{attribute 'linkalways'} 
{attribute 'no_explicit_call' := 'This FB is a CLASS and must be accessed using methods or properties'}
{attribute 'enable_dynamic_creation'}
FUNCTION_BLOCK Node_F_VN_ReadBarcodeExp2 EXTENDS VisionNode
VAR
    ipSrcImage : _ITcVnImage;
    ipDecodedData : _ITcVnContainer;
	ipContours : _ITcVnContainer;
    eBarcodeType : _ETcVnBarcodeType(ETcVnBarcodeType.TCVN_BT_ANY);
	nCodeNumber : _DINT(1);
	eSearchDirection : _ETcVnBarcodeSearchDirection(ETcVnBarcodeSearchDirection.TCVN_BSD_ANY);
	ipAngles : _ITcVnContainer; 
    hrPrev : _HRESULT(S_OK);
	hresult : _HRESULT(S_OK);
END_VAR

METHOD PUBLIC  Clone : I_Node
VAR
	pNode : POINTER TO Node_F_VN_ReadBarcodeExp2;
END_VAR
pNode := __NEW(Node_F_VN_ReadBarcodeExp2);
Clone := pNode^;
END_METHOD

METHOD FB_init : BOOL
VAR_INPUT
	bInitRetains : BOOL; // if TRUE, the retain variables are initialized (warm start / cold start)
	bInCopyCode : BOOL;  // if TRUE, the instance afterwards gets moved into the copy code (online change)
END_VAR
AddInput('ipSrcImage', ipSrcImage);
AddParameter('eBarcodeType', eBarcodeType);
AddParameter('nCodeNumber', nCodeNumber);
AddParameter('eSearchDirection', eSearchDirection);
AddInput('hrPrev', hrPrev);
AddOutput('ipDecodedData', ipDecodedData);
AddOutput('ipContours', ipContours);
AddOutput('ipAngles', ipAngles);
AddOutput('hresult',hresult);
END_METHOD

METHOD PROTECTED OnExecute
hresult.Value := F_VN_ReadBarcodeExp2(
	ipSrcImage := ipSrcImage.Value,
    ipDecodedData := ipDecodedData.Value,
	ipContours := ipContours.Value,
    eBarcodeType := eBarcodeType.Value,
	nCodeNumber := nCodeNumber.Value,
	eSearchDirection := eSearchDirection.Value,
	ipAngles := ipAngles.Value,
	hrPrev:= hrPrev.Value);
END_METHOD

METHOD PUBLIC PreExecutionCheck
VAR_INPUT
	Check : I_PreExecutionChecks;
END_VAR
Check.IsTrue(ipSrcImage.IsValid, 'ipSrcImage must contain an image');
Check.IsTrue((ipSrcImage.HasChannelCount(1) OR ipSrcImage.HasChannelCount(3)), 'ipSrcImage must have 1 or 3 channels');
Check.IsTrue(ipSrcImage.IsPixelDepth(8), 'ipSrcImage must have 8 bit pixel depth');
Check.IsTrue((nCodeNumber.Value = 1), 'nCodeNumber, currently only 1 supported');
END_METHOD

END_FUNCTION_BLOCK

(* stored: Version 1.1.0.1, ProductVersion 3.1.4026.13
   POU Node_F_VN_ReadBarcodeExp2: Id {65c1bd62-7353-0f6e-29a4-22a7e6e8fdd6}, SpecialFunc None
   Folder Constructor: Id {f820418b-973e-0913-0120-fec8fa28283e}
   Method Clone: Id {bd9e1304-df4e-0afa-28f3-b1ac6704a465}
   Method FB_init: Id {4f140e9f-790b-0b9a-2f98-55cfd4d8cc1f}
   Method OnExecute: Id {5058e32b-195d-0741-1701-339134b3d8a3}
   Method PreExecutionCheck: Id {18292969-6f49-0827-0306-dbc4ddbba5d9} *)
